{attribute 'Tc2GvlVarNames'}
VAR_CONFIG
END_VAR

(* stored: Version 1.1.0.1, ProductVersion 3.1.4018.9
   GVL Variable_Configuration: Id {7867c2d3-7ec9-4282-8299-ba884d68817c} *)
